{attribute 'qualified_only'}
{attribute 'strict'}
TYPE E_AssyState :
(
	PASS := 0,
	FAIL := 1,
	BREAK := 2
);
END_TYPE

(* stored: Version 1.1.0.1
   DUT E_AssyState: Id {f57b21b7-3460-048d-2d2c-ef8e35cdcd67} *)
